(* Schneider Machine Expert - Basic project MOTOR-START-DELTA, file version 1.7.0.0 *)
(* ProjectInformations: Name=New project *)

HARDWARE
  Cpu 0: TM221ME16R/G
  EthernetConfiguration: NetworkName=M221, IpAllocationMode=FixedAddress, IpAddress=0.0.0.0, SubnetMask=0.0.0.0
  SerialLineConfiguration: Baud=Baud19200, Parity=ParityEven, DataBits=DataBits8, StopBits=StopBits1, PhysicalMedium=PhysicalMediumRs485, TransmissionMode=TransmissionModeModbusRtu, SlaveId=1, Addressing=SlaveAddressing
  MastTask: UsePeriodScanMode=false, PeriodScan=100
  FastTask: Period=255
  CpuBehavior: StartingMode=StartAsPreviousState, AutoSaveRamOnEeprom=true, WatchdogPeriod=250

SYMBOLS  (address, symbol, comment, settings)
  %M0         "MEMO1"
  %M1         "MEMO2"
  %TM0        "TIMER"  [Preset=15, Base=OneSecond, IsRetentive=true]
  %I0.0       "SW1"
  %I0.1       "SW2"
  %Q0.0       "K1M"
  %Q0.1       "K2M"
  %Q0.2       "K3M"
  %Q0.3       "L1"
  %Q0.4       "L2"

POU New POU
  (* SectionNumber=1 *)

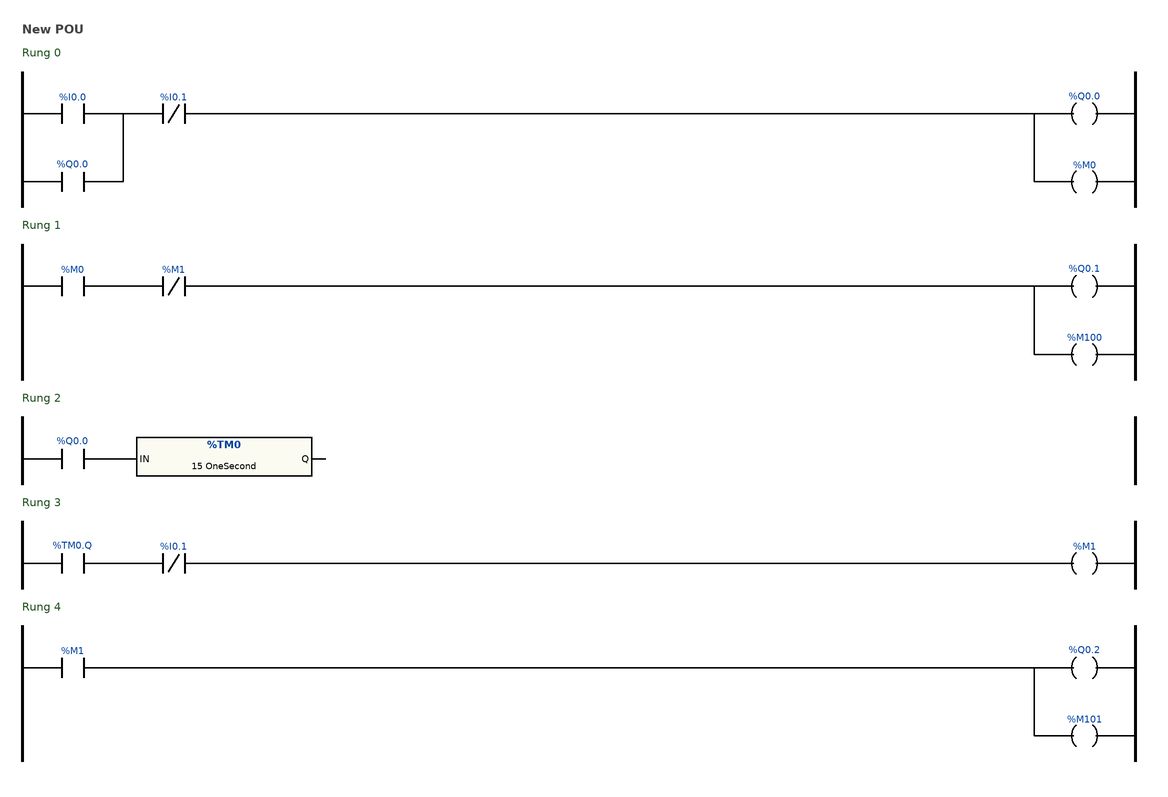

// Rung 0
  LD %I0.0
  OR %Q0.0
  ANDN %I0.1
  ST %Q0.0
  ST %M0
  // as ST:
  //   _t1 := (%I0.0 OR %Q0.0) AND NOT %I0.1;
  //   %Q0.0 := _t1;
  //   %M0 := _t1;

// Rung 1
  LD %M0
  ANDN %M1
  ST %Q0.1
  ST %M100
  // as ST:
  //   %Q0.1 := %M0 AND NOT %M1;
  //   %M100 := %M0 AND NOT %M1;

// Rung 2
  BLK %TM0
  LD %Q0.0
  IN
  END_BLK
  // as ST:
  //   %TM0(IN := %Q0.0);

// Rung 3
  LD %TM0.Q
  ANDN %I0.1
  ST %M1
  // as ST:
  //   %M1 := %TM0.Q AND NOT %I0.1;

// Rung 4
  LD %M1
  ST %Q0.2
  ST %M101
  // as ST:
  //   %Q0.2 := %M1;
  //   %M101 := %M1;
